// TIA Portal project "Scene_3" (V17)

(* hardware
DEVICE "S71500/ET200MP-Station_1"  S7-1500 station
   slot 0: "Profilschiene_0"  6ES7 590-1***0-0AA0
   slot 1: "PLC_1"  CPU 1511-1 PN  6ES7 511-1AK00-0AB0  V1.8
   slot 2: "AI 8xU/I/RTD/TC ST_1"  AI 8xU/I/RTD/TC ST  6ES7 531-7KF00-0AB0  V2.0
   slot 3: "AI 8xU/I/RTD/TC ST_2"  AI 8xU/I/RTD/TC ST  6ES7 531-7KF00-0AB0  V2.0
   slot 4: "AI 8xU/I/RTD/TC ST_3"  AI 8xU/I/RTD/TC ST  6ES7 531-7KF00-0AB0  V2.0
   slot 5: "AI 8xU/I/RTD/TC ST_4"  AI 8xU/I/RTD/TC ST  6ES7 531-7KF00-0AB0  V2.0
   slot 6: "DI 16x24VDC BA_1"  DI 16x24VDC BA  6ES7 521-1BH10-0AA0  V1.0
*)

// ===== PLC "PLC_1"  CPU 1511-1 PN =====

VAR_GLOBAL   // PLC tag table "Standard-Variablentabelle"
   "Fill" AT %I0.0 : Bool;
   "Discharge" AT %I0.1 : Bool;
   "Fill_valve" AT %Q0.0 : Bool;
   "Filling" AT %Q0.1 : Bool;
   "Discharge_valve" AT %Q0.2 : Bool;
   "Discharging_valve" AT %Q0.3 : Bool;
   "tag_1" AT %M0.0 : Bool;
   "tag_2" AT %M0.1 : Bool;
END_VAR

FUNCTION "MHJ-PLC-Lab-Function-S71500" : Void   // FC9000, SCL
{ S7_Optimized_Access := 'TRUE' }
VERSION : 0.1
   VAR_TEMP
      Value : Byte;
      ForCounter : Int;
   END_VAR
   VAR CONSTANT
      Value_01_DW : DWord := 16#1223_5486;
      Value_02_DW : DWord := 16#A6C9_D1F5;
   END_VAR
BEGIN

   #Value:=PEEK(area := 16#82,
        dbNumber := 0,
        byteOffset := 511);
   #Value := #Value + 1;

   POKE(area := 16#82,
        dbNumber := 0,
        byteOffset := 511,
        value := #Value);

   POKE(area := 16#82,
        dbNumber := 0,
        byteOffset := 1016,
        value := #Value_01_DW);
   POKE(area := 16#82,
        dbNumber := 0,
        byteOffset := 1020,
        value := #Value_02_DW);

   FOR #ForCounter := 0 TO 63 DO
       #Value:=PEEK(area := 16#1,
            dbNumber := 0,
            byteOffset := #ForCounter);
       POKE(area := 16#81,
            dbNumber := 0,
            byteOffset := #ForCounter,
            value := #Value);
   END_FOR;
   #Value := PEEK(area := 16#1,
                  dbNumber := 0,
                  byteOffset := 512);
   POKE(area := 16#82,
        dbNumber := 0,
        byteOffset := 512,
        value := #Value);
END_FUNCTION

ORGANIZATION_BLOCK "Main"   // OB1, LAD, ProgramCycle
TITLE = "Main Program Sweep (Cycle)"
{ S7_Optimized_Access := 'TRUE' }
VERSION : 0.1
   VAR_INPUT
      Initial_Call : Bool;   // Initial call of this OB
      Remanence : Bool;   // =True, if remanent data are available
   END_VAR
   VAR_TEMP   // added for the SCL form of the ladder/FBD networks
      _w1 : Bool;
      _w2 : Bool;
   END_VAR
BEGIN

REGION Network 1: Connection to Factory I/O
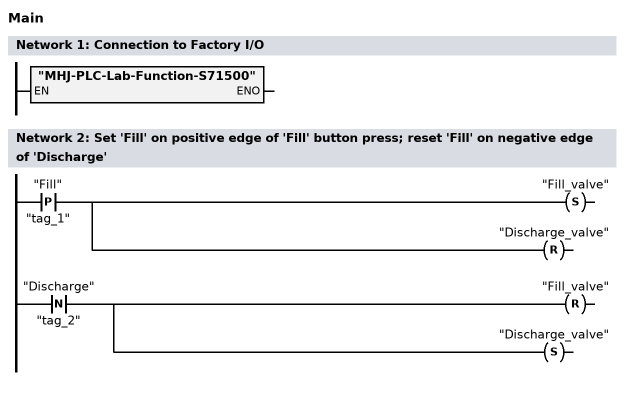
   RUNG wire#powerrail
      "MHJ-PLC-Lab-Function-S71500"()
   END_RUNG
   // the same network as SCL:
   "MHJ-PLC-Lab-Function-S71500"();
END_REGION

REGION Network 2: Set 'Fill' on positive edge of 'Fill' button press; reset 'Fill' on negative edge of 'Discharge'
   RUNG wire#powerrail
      P_Contact(operand := "Fill", bit := "tag_1")
      wire#w1
      S_Coil( "Fill_valve" )
   END_RUNG
   RUNG wire#w1
      R_Coil( "Discharge_valve" )
   END_RUNG
   RUNG wire#powerrail
      N_Contact(operand := "Discharge", bit := "tag_2")
      wire#w2
      R_Coil( "Fill_valve" )
   END_RUNG
   RUNG wire#w2
      S_Coil( "Discharge_valve" )
   END_RUNG
   // the same network as SCL:
   #_w1 := "Fill" AND NOT "tag_1";   // rising edge of "Fill"
   "tag_1" := "Fill";
   IF #_w1 THEN
       "Fill_valve" := TRUE;
       "Discharge_valve" := FALSE;
   END_IF;
   #_w2 := NOT "Discharge" AND "tag_2";   // falling edge of "Discharge"
   "tag_2" := "Discharge";
   IF #_w2 THEN
       "Fill_valve" := FALSE;
       "Discharge_valve" := TRUE;
   END_IF;
END_REGION
END_ORGANIZATION_BLOCK